Staubli VAL3: SetFrame.pgx

public program SetFrame(string x_sFrame (dimensions=1))
begin
  //
  sFrameName=x_sFrame
end
